// TwinCAT 3 PLC project TcUnit_Tests
// ProgramVersion: 3.1.4024.12
// libraries:
//   Tc2_Standard, * (Beckhoff Automation GmbH)
//   Tc2_System, * (Beckhoff Automation GmbH)
//   Tc3_Module, * (Beckhoff Automation GmbH)
//   TcUnit, * (www.tcunit.org)
// project tree:
//   / PlcTask.TcTTO (not stored)
//   POUs/ FB_FanControl.TcPOU (not stored), FC_HeatingCurve.TcPOU (not stored)
//   Test/ FB_FanControl_Test.TcPOU, FC_HeatingCurve_Test.TcPOU (not stored), PRG_TEST.TcPOU
// real-time tasks:
//   TASK PlcTask: cycle T#10ms, priority 20, ADS port 350

// ---- Test/FB_FanControl_Test.TcPOU
FUNCTION_BLOCK FB_FanControl_Test EXTENDS FB_TestSuite
VAR
END_VAR

FanSpeedMax();
FanSpeedZero();

METHOD FanSpeedMax
VAR
	fbFanControl : FB_FanControl;		//Function Block call
	FanControlRes : INT;				//Actual value of FanControl
	ExpectedValue : INT := 32767;		//Expected value for FanControl
END_VAR
TEST('FanSpeedMax');
 
fbFanControl.fSpeed := 100;
fbFanControl();
FanControlRes := fbFanControl.fSpeedSetRaw;
 
AssertEquals(Expected := ExpectedValue,
             Actual := FanControlRes,
             Message := 'The calculation is not correct');
 
TEST_FINISHED();
END_METHOD

METHOD FanSpeedZero
VAR
	fbFanControl : FB_FanControl;		//Function Block call
	FanControlRes : INT;				//Actual value of FanControl
	ExpectedValue : INT := 0;			//Expected value for FanControl

END_VAR
TEST('FanSpeedZero');
 
fbFanControl.fSpeed := 0;
fbFanControl();
FanControlRes := fbFanControl.fSpeedSetRaw;
 
AssertEquals(Expected := ExpectedValue,
             Actual := FanControlRes,
             Message := 'The calculation is not correct');
 
TEST_FINISHED();
END_METHOD

END_FUNCTION_BLOCK

// ---- Test/PRG_TEST.TcPOU
PROGRAM PRG_TEST
VAR
	HeatingCurve_Test : FC_HeatingCurve_Test;
	FanControlTest : FB_FanControl_Test;
END_VAR

TcUnit.RUN();

END_PROGRAM
